TYPE ZData :
STRUCT
  Config : ZDataConfig;
  Machine : ZDataMachine;
  Calibration : ZDataCalibration;
  Recipe : ZDataRecipe;
END_STRUCT
END_TYPE

(* stored: Version 1.1.0.1
   DUT ZData: Id {b64407f5-af9b-4462-86ec-1e8302a1bd38} *)
